FUNCTION TFNumeroPacchiSuLinea : UINT
VAR_INPUT
	ArrayPacchi : POINTER TO DUT_ArrayPacchi; 					//Array contenente i pacchi sui trasporti				
END_VAR
VAR
	i : UINT;
//	j : uint;
END_VAR

TFNumeroPacchiSuLinea := 0; 

FOR i:= 1 TO MAXDIMARRAYPACCHI DO
	//FOR j:= 1 TO MAXHANDLINGPACK-1 DO
		IF ArrayPacchi^.Pacco[i].ID.ID_Pacco[0] > 0 THEN
			TFNumeroPacchiSuLinea := TFNumeroPacchiSuLinea +1;
		END_IF
	//END_FOR
END_FOR

END_FUNCTION

(* stored: Version 1.1.0.1, ProductVersion 3.1.4024.11
   POU TFNumeroPacchiSuLinea: Id {8f764da7-feb1-47a2-9b06-9bacd2aaaa80}, SpecialFunc None *)
